FUNCTION_BLOCK NOT10 (* Basic Function Block Type *)
  (* Standard: 61499-2 *)
  (* Version 0.0, 9/18/2014, Администратор, nxtControl GmbH, Template *)
  PACKAGE Main;
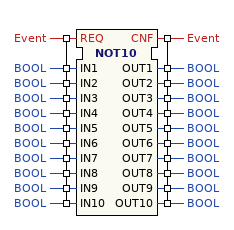
  EVENT_INPUT
    REQ WITH IN1, IN2, IN3, IN4, IN5, IN6, IN7, IN8, IN9, IN10; (* Normal Execution Request *)
  END_EVENT
  EVENT_OUTPUT
    CNF WITH OUT1, OUT2, OUT3, OUT4, OUT5, OUT6, OUT7, OUT8, OUT9, OUT10; (* Execution Confirmation *)
  END_EVENT
  VAR_INPUT
    IN1 : BOOL; (* Input event qualifier *)
    IN2 : BOOL;
    IN3 : BOOL;
    IN4 : BOOL;
    IN5 : BOOL;
    IN6 : BOOL;
    IN7 : BOOL;
    IN8 : BOOL;
    IN9 : BOOL;
    IN10 : BOOL;
  END_VAR
  VAR_OUTPUT
    OUT1 : BOOL; (* Output event qualifier *)
    OUT2 : BOOL;
    OUT3 : BOOL;
    OUT4 : BOOL;
    OUT5 : BOOL;
    OUT6 : BOOL;
    OUT7 : BOOL;
    OUT8 : BOOL;
    OUT9 : BOOL;
    OUT10 : BOOL;
  END_VAR
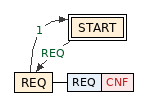
  EC_STATES
    START; (* Initial State *)
    REQ : REQ -> CNF; (* Normal execution *)
  END_STATES
  EC_TRANSITIONS
    START TO REQ := REQ;
    REQ TO START := 1;
  END_TRANSITIONS
  ALGORITHM REQ IN ST:
OUT1 := NOT IN1;
OUT2 := NOT IN2;
OUT3 := NOT IN3;
OUT4 := NOT IN4;
OUT5 := NOT IN5;
OUT6 := NOT IN6;
OUT7 := NOT IN7;
OUT8 := NOT IN8;
OUT9 := NOT IN9;
OUT10 := NOT IN10;
  END_ALGORITHM
END_FUNCTION_BLOCK
